TYPE ST_VRC_NO EXTENDS ST_ValveBase:
STRUCT
(* Readbacks *)
    //In case VRC is normally open
    {attribute 'pytmc' := '
    pv: CLS_OK;
    field: ONAM TRUE;
    field: ZNAM FALSE;
    io: i;
    '}
    xCLS_OK : BOOL := TRUE;
    {attribute 'pytmc' := '
    pv: CLS_SW ;
    field: ONAM CLOSE;
    field: ZNAM OPEN;
    io: io ;
    '}
    pv_xCLS_SW	: BOOL;

    {attribute 'pytmc' := '
    pv: CLS_DO ;
    field: ONAM CLOSE;
    field: ZNAM OPEN;
    io: io ;
    '}
    q_xCLS_DO	: BOOL;
    {attribute 'pytmc' := '
    pv: FORCE_CLS;
    field: ONAM FORCE CLOSE;
    field: ZNAM FALSE;
    io: io;
    '}
    pv_xOvrdCls	:	BOOL;

END_STRUCT
END_TYPE

(* stored: Version 1.1.0.1
   DUT ST_VRC_NO: Id {3c78b61e-192a-4faf-ac1e-61fc63c91393} *)
